    v3[14, 11] := "BsplineEval"(x := v0[11], lut_grid := "NeuroPLC_Weights".w0, lut_table := lut_tmp);
    // φ[12→14]: evaluate LUT (table offset 6060)
    FOR k := 0 TO 14 DO
        lut_tmp[k] := "NeuroPLC_Weights".w1[6060 + k];
    END_FOR;
    v3[14, 12] := "BsplineEval"(x := v0[12], lut_grid := "NeuroPLC_Weights".w0, lut_table := lut_tmp);
    // φ[13→14]: evaluate LUT (table offset 6075)
    FOR k := 0 TO 14 DO
        lut_tmp[k] := "NeuroPLC_Weights".w1[6075 + k];
    END_FOR;
    v3[14, 13] := "BsplineEval"(x := v0[13], lut_grid := "NeuroPLC_Weights".w0, lut_table := lut_tmp);
    // φ[14→14]: evaluate LUT (table offset 6090)
    FOR k := 0 TO 14 DO
        lut_tmp[k] := "NeuroPLC_Weights".w1[6090 + k];
    END_FOR;
    v3[14, 14] := "BsplineEval"(x := v0[14], lut_grid := "NeuroPLC_Weights".w0, lut_table := lut_tmp);
    // φ[15→14]: evaluate LUT (table offset 6105)
    FOR k := 0 TO 14 DO
        lut_tmp[k] := "NeuroPLC_Weights".w1[6105 + k];
    END_FOR;
    v3[14, 15] := "BsplineEval"(x := v0[15], lut_grid := "NeuroPLC_Weights".w0, lut_table := lut_tmp);
    // φ[16→14]: evaluate LUT (table offset 6120)
    FOR k := 0 TO 14 DO
        lut_tmp[k] := "NeuroPLC_Weights".w1[6120 + k];
    END_FOR;
    v3[14, 16] := "BsplineEval"(x := v0[16], lut_grid := "NeuroPLC_Weights".w0, lut_table := lut_tmp);
    // φ[17→14]: evaluate LUT (table offset 6135)
    FOR k := 0 TO 14 DO
        lut_tmp[k] := "NeuroPLC_Weights".w1[6135 + k];
    END_FOR;
    v3[14, 17] := "BsplineEval"(x := v0[17], lut_grid := "NeuroPLC_Weights".w0, lut_table := lut_tmp);
    // φ[18→14]: evaluate LUT (table offset 6150)
    FOR k := 0 TO 14 DO
        lut_tmp[k] := "NeuroPLC_Weights".w1[6150 + k];
    END_FOR;
    v3[14, 18] := "BsplineEval"(x := v0[18], lut_grid := "NeuroPLC_Weights".w0, lut_table := lut_tmp);
    // φ[19→14]: evaluate LUT (table offset 6165)
    FOR k := 0 TO 14 DO
        lut_tmp[k] := "NeuroPLC_Weights".w1[6165 + k];
    END_FOR;
    v3[14, 19] := "BsplineEval"(x := v0[19], lut_grid := "NeuroPLC_Weights".w0, lut_table := lut_tmp);
    // φ[20→14]: evaluate LUT (table offset 6180)
    FOR k := 0 TO 14 DO
        lut_tmp[k] := "NeuroPLC_Weights".w1[6180 + k];
    END_FOR;
    v3[14, 20] := "BsplineEval"(x := v0[20], lut_grid := "NeuroPLC_Weights".w0, lut_table := lut_tmp);
    // φ[21→14]: evaluate LUT (table offset 6195)
    FOR k := 0 TO 14 DO
        lut_tmp[k] := "NeuroPLC_Weights".w1[6195 + k];
    END_FOR;
    v3[14, 21] := "BsplineEval"(x := v0[21], lut_grid := "NeuroPLC_Weights".w0, lut_table := lut_tmp);
    // φ[22→14]: evaluate LUT (table offset 6210)
    FOR k := 0 TO 14 DO
        lut_tmp[k] := "NeuroPLC_Weights".w1[6210 + k];
    END_FOR;
    v3[14, 22] := "BsplineEval"(x := v0[22], lut_grid := "NeuroPLC_Weights".w0, lut_table := lut_tmp);
    // φ[23→14]: evaluate LUT (table offset 6225)
    FOR k := 0 TO 14 DO
        lut_tmp[k] := "NeuroPLC_Weights".w1[6225 + k];
    END_FOR;
    v3[14, 23] := "BsplineEval"(x := v0[23], lut_grid := "NeuroPLC_Weights".w0, lut_table := lut_tmp);
    // φ[24→14]: evaluate LUT (table offset 6240)
    FOR k := 0 TO 14 DO
        lut_tmp[k] := "NeuroPLC_Weights".w1[6240 + k];
    END_FOR;
    v3[14, 24] := "BsplineEval"(x := v0[24], lut_grid := "NeuroPLC_Weights".w0, lut_table := lut_tmp);
    // φ[25→14]: evaluate LUT (table offset 6255)
    FOR k := 0 TO 14 DO
        lut_tmp[k] := "NeuroPLC_Weights".w1[6255 + k];
    END_FOR;
    v3[14, 25] := "BsplineEval"(x := v0[25], lut_grid := "NeuroPLC_Weights".w0, lut_table := lut_tmp);
    // φ[26→14]: evaluate LUT (table offset 6270)
    FOR k := 0 TO 14 DO
        lut_tmp[k] := "NeuroPLC_Weights".w1[6270 + k];
    END_FOR;
    v3[14, 26] := "BsplineEval"(x := v0[26], lut_grid := "NeuroPLC_Weights".w0, lut_table := lut_tmp);
    // φ[27→14]: evaluate LUT (table offset 6285)
    FOR k := 0 TO 14 DO
        lut_tmp[k] := "NeuroPLC_Weights".w1[6285 + k];
    END_FOR;
    v3[14, 27] := "BsplineEval"(x := v0[27], lut_grid := "NeuroPLC_Weights".w0, lut_table := lut_tmp);
    // φ[0→15]: evaluate LUT (table offset 6300)
    FOR k := 0 TO 14 DO
        lut_tmp[k] := "NeuroPLC_Weights".w1[6300 + k];
    END_FOR;
    v3[15, 0] := "BsplineEval"(x := v0[0], lut_grid := "NeuroPLC_Weights".w0, lut_table := lut_tmp);
    // φ[1→15]: evaluate LUT (table offset 6315)
    FOR k := 0 TO 14 DO
        lut_tmp[k] := "NeuroPLC_Weights".w1[6315 + k];
    END_FOR;
    v3[15, 1] := "BsplineEval"(x := v0[1], lut_grid := "NeuroPLC_Weights".w0, lut_table := lut_tmp);
    // φ[2→15]: evaluate LUT (table offset 6330)
    FOR k := 0 TO 14 DO
        lut_tmp[k] := "NeuroPLC_Weights".w1[6330 + k];
    END_FOR;
    v3[15, 2] := "BsplineEval"(x := v0[2], lut_grid := "NeuroPLC_Weights".w0, lut_table := lut_tmp);
    // φ[3→15]: evaluate LUT (table offset 6345)
    FOR k := 0 TO 14 DO
        lut_tmp[k] := "NeuroPLC_Weights".w1[6345 + k];
    END_FOR;
    v3[15, 3] := "BsplineEval"(x := v0[3], lut_grid := "NeuroPLC_Weights".w0, lut_table := lut_tmp);
    // φ[4→15]: evaluate LUT (table offset 6360)
    FOR k := 0 TO 14 DO
        lut_tmp[k] := "NeuroPLC_Weights".w1[6360 + k];
    END_FOR;
    v3[15, 4] := "BsplineEval"(x := v0[4], lut_grid := "NeuroPLC_Weights".w0, lut_table := lut_tmp);
    // φ[5→15]: evaluate LUT (table offset 6375)
    FOR k := 0 TO 14 DO
        lut_tmp[k] := "NeuroPLC_Weights".w1[6375 + k];
    END_FOR;
    v3[15, 5] := "BsplineEval"(x := v0[5], lut_grid := "NeuroPLC_Weights".w0, lut_table := lut_tmp);
    // φ[6→15]: evaluate LUT (table offset 6390)
    FOR k := 0 TO 14 DO
        lut_tmp[k] := "NeuroPLC_Weights".w1[6390 + k];
    END_FOR;
    v3[15, 6] := "BsplineEval"(x := v0[6], lut_grid := "NeuroPLC_Weights".w0, lut_table := lut_tmp);
    // φ[7→15]: evaluate LUT (table offset 6405)
    FOR k := 0 TO 14 DO
        lut_tmp[k] := "NeuroPLC_Weights".w1[6405 + k];
    END_FOR;
    v3[15, 7] := "BsplineEval"(x := v0[7], lut_grid := "NeuroPLC_Weights".w0, lut_table := lut_tmp);
    // φ[8→15]: evaluate LUT (table offset 6420)
    FOR k := 0 TO 14 DO
        lut_tmp[k] := "NeuroPLC_Weights".w1[6420 + k];
    END_FOR;
    v3[15, 8] := "BsplineEval"(x := v0[8], lut_grid := "NeuroPLC_Weights".w0, lut_table := lut_tmp);
    // φ[9→15]: evaluate LUT (table offset 6435)
    FOR k := 0 TO 14 DO
        lut_tmp[k] := "NeuroPLC_Weights".w1[6435 + k];
    END_FOR;
    v3[15, 9] := "BsplineEval"(x := v0[9], lut_grid := "NeuroPLC_Weights".w0, lut_table := lut_tmp);
    // φ[10→15]: evaluate LUT (table offset 6450)
    FOR k := 0 TO 14 DO
        lut_tmp[k] := "NeuroPLC_Weights".w1[6450 + k];
    END_FOR;
    v3[15, 10] := "BsplineEval"(x := v0[10], lut_grid := "NeuroPLC_Weights".w0, lut_table := lut_tmp);
    // φ[11→15]: evaluate LUT (table offset 6465)
    FOR k := 0 TO 14 DO
        lut_tmp[k] := "NeuroPLC_Weights".w1[6465 + k];
    END_FOR;
    v3[15, 11] := "BsplineEval"(x := v0[11], lut_grid := "NeuroPLC_Weights".w0, lut_table := lut_tmp);
    // φ[12→15]: evaluate LUT (table offset 6480)
    FOR k := 0 TO 14 DO
        lut_tmp[k] := "NeuroPLC_Weights".w1[6480 + k];
    END_FOR;
    v3[15, 12] := "BsplineEval"(x := v0[12], lut_grid := "NeuroPLC_Weights".w0, lut_table := lut_tmp);
    // φ[13→15]: evaluate LUT (table offset 6495)
    FOR k := 0 TO 14 DO
        lut_tmp[k] := "NeuroPLC_Weights".w1[6495 + k];
    END_FOR;
    v3[15, 13] := "BsplineEval"(x := v0[13], lut_grid := "NeuroPLC_Weights".w0, lut_table := lut_tmp);
    // φ[14→15]: evaluate LUT (table offset 6510)
    FOR k := 0 TO 14 DO
        lut_tmp[k] := "NeuroPLC_Weights".w1[6510 + k];
    END_FOR;
    v3[15, 14] := "BsplineEval"(x := v0[14], lut_grid := "NeuroPLC_Weights".w0, lut_table := lut_tmp);
    // φ[15→15]: evaluate LUT (table offset 6525)
    FOR k := 0 TO 14 DO
        lut_tmp[k] := "NeuroPLC_Weights".w1[6525 + k];
    END_FOR;
    v3[15, 15] := "BsplineEval"(x := v0[15], lut_grid := "NeuroPLC_Weights".w0, lut_table := lut_tmp);
    // φ[16→15]: evaluate LUT (table offset 6540)
    FOR k := 0 TO 14 DO
        lut_tmp[k] := "NeuroPLC_Weights".w1[6540 + k];
    END_FOR;
    v3[15, 16] := "BsplineEval"(x := v0[16], lut_grid := "NeuroPLC_Weights".w0, lut_table := lut_tmp);
    // φ[17→15]: evaluate LUT (table offset 6555)
    FOR k := 0 TO 14 DO
        lut_tmp[k] := "NeuroPLC_Weights".w1[6555 + k];
    END_FOR;
    v3[15, 17] := "BsplineEval"(x := v0[17], lut_grid := "NeuroPLC_Weights".w0, lut_table := lut_tmp);
    // φ[18→15]: evaluate LUT (table offset 6570)
    FOR k := 0 TO 14 DO
        lut_tmp[k] := "NeuroPLC_Weights".w1[6570 + k];
    END_FOR;
    v3[15, 18] := "BsplineEval"(x := v0[18], lut_grid := "NeuroPLC_Weights".w0, lut_table := lut_tmp);
    // φ[19→15]: evaluate LUT (table offset 6585)
    FOR k := 0 TO 14 DO
        lut_tmp[k] := "NeuroPLC_Weights".w1[6585 + k];
    END_FOR;
    v3[15, 19] := "BsplineEval"(x := v0[19], lut_grid := "NeuroPLC_Weights".w0, lut_table := lut_tmp);
    // φ[20→15]: evaluate LUT (table offset 6600)
    FOR k := 0 TO 14 DO
        lut_tmp[k] := "NeuroPLC_Weights".w1[6600 + k];
    END_FOR;
    v3[15, 20] := "BsplineEval"(x := v0[20], lut_grid := "NeuroPLC_Weights".w0, lut_table := lut_tmp);
    // φ[21→15]: evaluate LUT (table offset 6615)
    FOR k := 0 TO 14 DO
        lut_tmp[k] := "NeuroPLC_Weights".w1[6615 + k];
    END_FOR;
    v3[15, 21] := "BsplineEval"(x := v0[21], lut_grid := "NeuroPLC_Weights".w0, lut_table := lut_tmp);
    // φ[22→15]: evaluate LUT (table offset 6630)
    FOR k := 0 TO 14 DO
        lut_tmp[k] := "NeuroPLC_Weights".w1[6630 + k];
    END_FOR;
    v3[15, 22] := "BsplineEval"(x := v0[22], lut_grid := "NeuroPLC_Weights".w0, lut_table := lut_tmp);
    // φ[23→15]: evaluate LUT (table offset 6645)
    FOR k := 0 TO 14 DO
        lut_tmp[k] := "NeuroPLC_Weights".w1[6645 + k];
    END_FOR;
    v3[15, 23] := "BsplineEval"(x := v0[23], lut_grid := "NeuroPLC_Weights".w0, lut_table := lut_tmp);
    // φ[24→15]: evaluate LUT (table offset 6660)
    FOR k := 0 TO 14 DO
        lut_tmp[k] := "NeuroPLC_Weights".w1[6660 + k];
    END_FOR;
    v3[15, 24] := "BsplineEval"(x := v0[24], lut_grid := "NeuroPLC_Weights".w0, lut_table := lut_tmp);
    // φ[25→15]: evaluate LUT (table offset 6675)
    FOR k := 0 TO 14 DO
        lut_tmp[k] := "NeuroPLC_Weights".w1[6675 + k];
    END_FOR;
    v3[15, 25] := "BsplineEval"(x := v0[25], lut_grid := "NeuroPLC_Weights".w0, lut_table := lut_tmp);
    // φ[26→15]: evaluate LUT (table offset 6690)
    FOR k := 0 TO 14 DO
        lut_tmp[k] := "NeuroPLC_Weights".w1[6690 + k];
    END_FOR;
    v3[15, 26] := "BsplineEval"(x := v0[26], lut_grid := "NeuroPLC_Weights".w0, lut_table := lut_tmp);
    // φ[27→15]: evaluate LUT (table offset 6705)
    FOR k := 0 TO 14 DO
        lut_tmp[k] := "NeuroPLC_Weights".w1[6705 + k];
    END_FOR;
    v3[15, 27] := "BsplineEval"(x := v0[27], lut_grid := "NeuroPLC_Weights".w0, lut_table := lut_tmp);

    // ---- l0_base: MatMul(28→16) ----
    // W = "NeuroPLC_Weights".w2[:448],   b = w2[448:]
    v2[0] := "NeuroPLC_Weights".w2[448 + 0] + "NeuroPLC_Weights".w2[0] * v1[0] + "NeuroPLC_Weights".w2[1] * v1[1] + "NeuroPLC_Weights".w2[2] * v1[2] + "NeuroPLC_Weights".w2[3] * v1[3] + "NeuroPLC_Weights".w2[4] * v1[4] + "NeuroPLC_Weights".w2[5] * v1[5] + "NeuroPLC_Weights".w2[6] * v1[6] + "NeuroPLC_Weights".w2[7] * v1[7] + "NeuroPLC_Weights".w2[8] * v1[8] + "NeuroPLC_Weights".w2[9] * v1[9] + "NeuroPLC_Weights".w2[10] * v1[10] + "NeuroPLC_Weights".w2[11] * v1[11] + "NeuroPLC_Weights".w2[12] * v1[12] + "NeuroPLC_Weights".w2[13] * v1[13] + "NeuroPLC_Weights".w2[14] * v1[14] + "NeuroPLC_Weights".w2[15] * v1[15] + "NeuroPLC_Weights".w2[16] * v1[16] + "NeuroPLC_Weights".w2[17] * v1[17] + "NeuroPLC_Weights".w2[18] * v1[18] + "NeuroPLC_Weights".w2[19] * v1[19] + "NeuroPLC_Weights".w2[20] * v1[20] + "NeuroPLC_Weights".w2[21] * v1[21] + "NeuroPLC_Weights".w2[22] * v1[22] + "NeuroPLC_Weights".w2[23] * v1[23] + "NeuroPLC_Weights".w2[24] * v1[24] + "NeuroPLC_Weights".w2[25] * v1[25] + "NeuroPLC_Weights".w2[26] * v1[26] + "NeuroPLC_Weights".w2[27] * v1[27];
    v2[1] := "NeuroPLC_Weights".w2[448 + 1] + "NeuroPLC_Weights".w2[28] * v1[0] + "NeuroPLC_Weights".w2[29] * v1[1] + "NeuroPLC_Weights".w2[30] * v1[2] + "NeuroPLC_Weights".w2[31] * v1[3] + "NeuroPLC_Weights".w2[32] * v1[4] + "NeuroPLC_Weights".w2[33] * v1[5] + "NeuroPLC_Weights".w2[34] * v1[6] + "NeuroPLC_Weights".w2[35] * v1[7] + "NeuroPLC_Weights".w2[36] * v1[8] + "NeuroPLC_Weights".w2[37] * v1[9] + "NeuroPLC_Weights".w2[38] * v1[10] + "NeuroPLC_Weights".w2[39] * v1[11] + "NeuroPLC_Weights".w2[40] * v1[12] + "NeuroPLC_Weights".w2[41] * v1[13] + "NeuroPLC_Weights".w2[42] * v1[14] + "NeuroPLC_Weights".w2[43] * v1[15] + "NeuroPLC_Weights".w2[44] * v1[16] + "NeuroPLC_Weights".w2[45] * v1[17] + "NeuroPLC_Weights".w2[46] * v1[18] + "NeuroPLC_Weights".w2[47] * v1[19] + "NeuroPLC_Weights".w2[48] * v1[20] + "NeuroPLC_Weights".w2[49] * v1[21] + "NeuroPLC_Weights".w2[50] * v1[22] + "NeuroPLC_Weights".w2[51] * v1[23] + "NeuroPLC_Weights".w2[52] * v1[24] + "NeuroPLC_Weights".w2[53] * v1[25] + "NeuroPLC_Weights".w2[54] * v1[26] + "NeuroPLC_Weights".w2[55] * v1[27];
    v2[2] := "NeuroPLC_Weights".w2[448 + 2] + "NeuroPLC_Weights".w2[56] * v1[0] + "NeuroPLC_Weights".w2[57] * v1[1] + "NeuroPLC_Weights".w2[58] * v1[2] + "NeuroPLC_Weights".w2[59] * v1[3] + "NeuroPLC_Weights".w2[60] * v1[4] + "NeuroPLC_Weights".w2[61] * v1[5] + "NeuroPLC_Weights".w2[62] * v1[6] + "NeuroPLC_Weights".w2[63] * v1[7] + "NeuroPLC_Weights".w2[64] * v1[8] + "NeuroPLC_Weights".w2[65] * v1[9] + "NeuroPLC_Weights".w2[66] * v1[10] + "NeuroPLC_Weights".w2[67] * v1[11] + "NeuroPLC_Weights".w2[68] * v1[12] + "NeuroPLC_Weights".w2[69] * v1[13] + "NeuroPLC_Weights".w2[70] * v1[14] + "NeuroPLC_Weights".w2[71] * v1[15] + "NeuroPLC_Weights".w2[72] * v1[16] + "NeuroPLC_Weights".w2[73] * v1[17] + "NeuroPLC_Weights".w2[74] * v1[18] + "NeuroPLC_Weights".w2[75] * v1[19] + "NeuroPLC_Weights".w2[76] * v1[20] + "NeuroPLC_Weights".w2[77] * v1[21] + "NeuroPLC_Weights".w2[78] * v1[22] + "NeuroPLC_Weights".w2[79] * v1[23] + "NeuroPLC_Weights".w2[80] * v1[24] + "NeuroPLC_Weights".w2[81] * v1[25] + "NeuroPLC_Weights".w2[82] * v1[26] + "NeuroPLC_Weights".w2[83] * v1[27];
    v2[3] := "NeuroPLC_Weights".w2[448 + 3] + "NeuroPLC_Weights".w2[84] * v1[0] + "NeuroPLC_Weights".w2[85] * v1[1] + "NeuroPLC_Weights".w2[86] * v1[2] + "NeuroPLC_Weights".w2[87] * v1[3] + "NeuroPLC_Weights".w2[88] * v1[4] + "NeuroPLC_Weights".w2[89] * v1[5] + "NeuroPLC_Weights".w2[90] * v1[6] + "NeuroPLC_Weights".w2[91] * v1[7] + "NeuroPLC_Weights".w2[92] * v1[8] + "NeuroPLC_Weights".w2[93] * v1[9] + "NeuroPLC_Weights".w2[94] * v1[10] + "NeuroPLC_Weights".w2[95] * v1[11] + "NeuroPLC_Weights".w2[96] * v1[12] + "NeuroPLC_Weights".w2[97] * v1[13] + "NeuroPLC_Weights".w2[98] * v1[14] + "NeuroPLC_Weights".w2[99] * v1[15] + "NeuroPLC_Weights".w2[100] * v1[16] + "NeuroPLC_Weights".w2[101] * v1[17] + "NeuroPLC_Weights".w2[102] * v1[18] + "NeuroPLC_Weights".w2[103] * v1[19] + "NeuroPLC_Weights".w2[104] * v1[20] + "NeuroPLC_Weights".w2[105] * v1[21] + "NeuroPLC_Weights".w2[106] * v1[22] + "NeuroPLC_Weights".w2[107] * v1[23] + "NeuroPLC_Weights".w2[108] * v1[24] + "NeuroPLC_Weights".w2[109] * v1[25] + "NeuroPLC_Weights".w2[110] * v1[26] + "NeuroPLC_Weights".w2[111] * v1[27];
    v2[4] := "NeuroPLC_Weights".w2[448 + 4] + "NeuroPLC_Weights".w2[112] * v1[0] + "NeuroPLC_Weights".w2[113] * v1[1] + "NeuroPLC_Weights".w2[114] * v1[2] + "NeuroPLC_Weights".w2[115] * v1[3] + "NeuroPLC_Weights".w2[116] * v1[4] + "NeuroPLC_Weights".w2[117] * v1[5] + "NeuroPLC_Weights".w2[118] * v1[6] + "NeuroPLC_Weights".w2[119] * v1[7] + "NeuroPLC_Weights".w2[120] * v1[8] + "NeuroPLC_Weights".w2[121] * v1[9] + "NeuroPLC_Weights".w2[122] * v1[10] + "NeuroPLC_Weights".w2[123] * v1[11] + "NeuroPLC_Weights".w2[124] * v1[12] + "NeuroPLC_Weights".w2[125] * v1[13] + "NeuroPLC_Weights".w2[126] * v1[14] + "NeuroPLC_Weights".w2[127] * v1[15] + "NeuroPLC_Weights".w2[128] * v1[16] + "NeuroPLC_Weights".w2[129] * v1[17] + "NeuroPLC_Weights".w2[130] * v1[18] + "NeuroPLC_Weights".w2[131] * v1[19] + "NeuroPLC_Weights".w2[132] * v1[20] + "NeuroPLC_Weights".w2[133] * v1[21] + "NeuroPLC_Weights".w2[134] * v1[22] + "NeuroPLC_Weights".w2[135] * v1[23] + "NeuroPLC_Weights".w2[136] * v1[24] + "NeuroPLC_Weights".w2[137] * v1[25] + "NeuroPLC_Weights".w2[138] * v1[26] + "NeuroPLC_Weights".w2[139] * v1[27];
    v2[5] := "NeuroPLC_Weights".w2[448 + 5] + "NeuroPLC_Weights".w2[140] * v1[0] + "NeuroPLC_Weights".w2[141] * v1[1] + "NeuroPLC_Weights".w2[142] * v1[2] + "NeuroPLC_Weights".w2[143] * v1[3] + "NeuroPLC_Weights".w2[144] * v1[4] + "NeuroPLC_Weights".w2[145] * v1[5] + "NeuroPLC_Weights".w2[146] * v1[6] + "NeuroPLC_Weights".w2[147] * v1[7] + "NeuroPLC_Weights".w2[148] * v1[8] + "NeuroPLC_Weights".w2[149] * v1[9] + "NeuroPLC_Weights".w2[150] * v1[10] + "NeuroPLC_Weights".w2[151] * v1[11] + "NeuroPLC_Weights".w2[152] * v1[12] + "NeuroPLC_Weights".w2[153] * v1[13] + "NeuroPLC_Weights".w2[154] * v1[14] + "NeuroPLC_Weights".w2[155] * v1[15] + "NeuroPLC_Weights".w2[156] * v1[16] + "NeuroPLC_Weights".w2[157] * v1[17] + "NeuroPLC_Weights".w2[158] * v1[18] + "NeuroPLC_Weights".w2[159] * v1[19] + "NeuroPLC_Weights".w2[160] * v1[20] + "NeuroPLC_Weights".w2[161] * v1[21] + "NeuroPLC_Weights".w2[162] * v1[22] + "NeuroPLC_Weights".w2[163] * v1[23] + "NeuroPLC_Weights".w2[164] * v1[24] + "NeuroPLC_Weights".w2[165] * v1[25] + "NeuroPLC_Weights".w2[166] * v1[26] + "NeuroPLC_Weights".w2[167] * v1[27];
    v2[6] := "NeuroPLC_Weights".w2[448 + 6] + "NeuroPLC_Weights".w2[168] * v1[0] + "NeuroPLC_Weights".w2[169] * v1[1] + "NeuroPLC_Weights".w2[170] * v1[2] + "NeuroPLC_Weights".w2[171] * v1[3] + "NeuroPLC_Weights".w2[172] * v1[4] + "NeuroPLC_Weights".w2[173] * v1[5] + "NeuroPLC_Weights".w2[174] * v1[6] + "NeuroPLC_Weights".w2[175] * v1[7] + "NeuroPLC_Weights".w2[176] * v1[8] + "NeuroPLC_Weights".w2[177] * v1[9] + "NeuroPLC_Weights".w2[178] * v1[10] + "NeuroPLC_Weights".w2[179] * v1[11] + "NeuroPLC_Weights".w2[180] * v1[12] + "NeuroPLC_Weights".w2[181] * v1[13] + "NeuroPLC_Weights".w2[182] * v1[14] + "NeuroPLC_Weights".w2[183] * v1[15] + "NeuroPLC_Weights".w2[184] * v1[16] + "NeuroPLC_Weights".w2[185] * v1[17] + "NeuroPLC_Weights".w2[186] * v1[18] + "NeuroPLC_Weights".w2[187] * v1[19] + "NeuroPLC_Weights".w2[188] * v1[20] + "NeuroPLC_Weights".w2[189] * v1[21] + "NeuroPLC_Weights".w2[190] * v1[22] + "NeuroPLC_Weights".w2[191] * v1[23] + "NeuroPLC_Weights".w2[192] * v1[24] + "NeuroPLC_Weights".w2[193] * v1[25] + "NeuroPLC_Weights".w2[194] * v1[26] + "NeuroPLC_Weights".w2[195] * v1[27];
    v2[7] := "NeuroPLC_Weights".w2[448 + 7] + "NeuroPLC_Weights".w2[196] * v1[0] + "NeuroPLC_Weights".w2[197] * v1[1] + "NeuroPLC_Weights".w2[198] * v1[2] + "NeuroPLC_Weights".w2[199] * v1[3] + "NeuroPLC_Weights".w2[200] * v1[4] + "NeuroPLC_Weights".w2[201] * v1[5] + "NeuroPLC_Weights".w2[202] * v1[6] + "NeuroPLC_Weights".w2[203] * v1[7] + "NeuroPLC_Weights".w2[204] * v1[8] + "NeuroPLC_Weights".w2[205] * v1[9] + "NeuroPLC_Weights".w2[206] * v1[10] + "NeuroPLC_Weights".w2[207] * v1[11] + "NeuroPLC_Weights".w2[208] * v1[12] + "NeuroPLC_Weights".w2[209] * v1[13] + "NeuroPLC_Weights".w2[210] * v1[14] + "NeuroPLC_Weights".w2[211] * v1[15] + "NeuroPLC_Weights".w2[212] * v1[16] + "NeuroPLC_Weights".w2[213] * v1[17] + "NeuroPLC_Weights".w2[214] * v1[18] + "NeuroPLC_Weights".w2[215] * v1[19] + "NeuroPLC_Weights".w2[216] * v1[20] + "NeuroPLC_Weights".w2[217] * v1[21] + "NeuroPLC_Weights".w2[218] * v1[22] + "NeuroPLC_Weights".w2[219] * v1[23] + "NeuroPLC_Weights".w2[220] * v1[24] + "NeuroPLC_Weights".w2[221] * v1[25] + "NeuroPLC_Weights".w2[222] * v1[26] + "NeuroPLC_Weights".w2[223] * v1[27];
    v2[8] := "NeuroPLC_Weights".w2[448 + 8] + "NeuroPLC_Weights".w2[224] * v1[0] + "NeuroPLC_Weights".w2[225] * v1[1] + "NeuroPLC_Weights".w2[226] * v1[2] + "NeuroPLC_Weights".w2[227] * v1[3] + "NeuroPLC_Weights".w2[228] * v1[4] + "NeuroPLC_Weights".w2[229] * v1[5] + "NeuroPLC_Weights".w2[230] * v1[6] + "NeuroPLC_Weights".w2[231] * v1[7] + "NeuroPLC_Weights".w2[232] * v1[8] + "NeuroPLC_Weights".w2[233] * v1[9] + "NeuroPLC_Weights".w2[234] * v1[10] + "NeuroPLC_Weights".w2[235] * v1[11] + "NeuroPLC_Weights".w2[236] * v1[12] + "NeuroPLC_Weights".w2[237] * v1[13] + "NeuroPLC_Weights".w2[238] * v1[14] + "NeuroPLC_Weights".w2[239] * v1[15] + "NeuroPLC_Weights".w2[240] * v1[16] + "NeuroPLC_Weights".w2[241] * v1[17] + "NeuroPLC_Weights".w2[242] * v1[18] + "NeuroPLC_Weights".w2[243] * v1[19] + "NeuroPLC_Weights".w2[244] * v1[20] + "NeuroPLC_Weights".w2[245] * v1[21] + "NeuroPLC_Weights".w2[246] * v1[22] + "NeuroPLC_Weights".w2[247] * v1[23] + "NeuroPLC_Weights".w2[248] * v1[24] + "NeuroPLC_Weights".w2[249] * v1[25] + "NeuroPLC_Weights".w2[250] * v1[26] + "NeuroPLC_Weights".w2[251] * v1[27];
    v2[9] := "NeuroPLC_Weights".w2[448 + 9] + "NeuroPLC_Weights".w2[252] * v1[0] + "NeuroPLC_Weights".w2[253] * v1[1] + "NeuroPLC_Weights".w2[254] * v1[2] + "NeuroPLC_Weights".w2[255] * v1[3] + "NeuroPLC_Weights".w2[256] * v1[4] + "NeuroPLC_Weights".w2[257] * v1[5] + "NeuroPLC_Weights".w2[258] * v1[6] + "NeuroPLC_Weights".w2[259] * v1[7] + "NeuroPLC_Weights".w2[260] * v1[8] + "NeuroPLC_Weights".w2[261] * v1[9] + "NeuroPLC_Weights".w2[262] * v1[10] + "NeuroPLC_Weights".w2[263] * v1[11] + "NeuroPLC_Weights".w2[264] * v1[12] + "NeuroPLC_Weights".w2[265] * v1[13] + "NeuroPLC_Weights".w2[266] * v1[14] + "NeuroPLC_Weights".w2[267] * v1[15] + "NeuroPLC_Weights".w2[268] * v1[16] + "NeuroPLC_Weights".w2[269] * v1[17] + "NeuroPLC_Weights".w2[270] * v1[18] + "NeuroPLC_Weights".w2[271] * v1[19] + "NeuroPLC_Weights".w2[272] * v1[20] + "NeuroPLC_Weights".w2[273] * v1[21] + "NeuroPLC_Weights".w2[274] * v1[22] + "NeuroPLC_Weights".w2[275] * v1[23] + "NeuroPLC_Weights".w2[276] * v1[24] + "NeuroPLC_Weights".w2[277] * v1[25] + "NeuroPLC_Weights".w2[278] * v1[26] + "NeuroPLC_Weights".w2[279] * v1[27];
    v2[10] := "NeuroPLC_Weights".w2[448 + 10] + "NeuroPLC_Weights".w2[280] * v1[0] + "NeuroPLC_Weights".w2[281] * v1[1] + "NeuroPLC_Weights".w2[282] * v1[2] + "NeuroPLC_Weights".w2[283] * v1[3] + "NeuroPLC_Weights".w2[284] * v1[4] + "NeuroPLC_Weights".w2[285] * v1[5] + "NeuroPLC_Weights".w2[286] * v1[6] + "NeuroPLC_Weights".w2[287] * v1[7] + "NeuroPLC_Weights".w2[288] * v1[8] + "NeuroPLC_Weights".w2[289] * v1[9] + "NeuroPLC_Weights".w2[290] * v1[10] + "NeuroPLC_Weights".w2[291] * v1[11] + "NeuroPLC_Weights".w2[292] * v1[12] + "NeuroPLC_Weights".w2[293] * v1[13] + "NeuroPLC_Weights".w2[294] * v1[14] + "NeuroPLC_Weights".w2[295] * v1[15] + "NeuroPLC_Weights".w2[296] * v1[16] + "NeuroPLC_Weights".w2[297] * v1[17] + "NeuroPLC_Weights".w2[298] * v1[18] + "NeuroPLC_Weights".w2[299] * v1[19] + "NeuroPLC_Weights".w2[300] * v1[20] + "NeuroPLC_Weights".w2[301] * v1[21] + "NeuroPLC_Weights".w2[302] * v1[22] + "NeuroPLC_Weights".w2[303] * v1[23] + "NeuroPLC_Weights".w2[304] * v1[24] + "NeuroPLC_Weights".w2[305] * v1[25] + "NeuroPLC_Weights".w2[306] * v1[26] + "NeuroPLC_Weights".w2[307] * v1[27];
    v2[11] := "NeuroPLC_Weights".w2[448 + 11] + "NeuroPLC_Weights".w2[308] * v1[0] + "NeuroPLC_Weights".w2[309] * v1[1] + "NeuroPLC_Weights".w2[310] * v1[2] + "NeuroPLC_Weights".w2[311] * v1[3] + "NeuroPLC_Weights".w2[312] * v1[4] + "NeuroPLC_Weights".w2[313] * v1[5] + "NeuroPLC_Weights".w2[314] * v1[6] + "NeuroPLC_Weights".w2[315] * v1[7] + "NeuroPLC_Weights".w2[316] * v1[8] + "NeuroPLC_Weights".w2[317] * v1[9] + "NeuroPLC_Weights".w2[318] * v1[10] + "NeuroPLC_Weights".w2[319] * v1[11] + "NeuroPLC_Weights".w2[320] * v1[12] + "NeuroPLC_Weights".w2[321] * v1[13] + "NeuroPLC_Weights".w2[322] * v1[14] + "NeuroPLC_Weights".w2[323] * v1[15] + "NeuroPLC_Weights".w2[324] * v1[16] + "NeuroPLC_Weights".w2[325] * v1[17] + "NeuroPLC_Weights".w2[326] * v1[18] + "NeuroPLC_Weights".w2[327] * v1[19] + "NeuroPLC_Weights".w2[328] * v1[20] + "NeuroPLC_Weights".w2[329] * v1[21] + "NeuroPLC_Weights".w2[330] * v1[22] + "NeuroPLC_Weights".w2[331] * v1[23] + "NeuroPLC_Weights".w2[332] * v1[24] + "NeuroPLC_Weights".w2[333] * v1[25] + "NeuroPLC_Weights".w2[334] * v1[26] + "NeuroPLC_Weights".w2[335] * v1[27];
    v2[12] := "NeuroPLC_Weights".w2[448 + 12] + "NeuroPLC_Weights".w2[336] * v1[0] + "NeuroPLC_Weights".w2[337] * v1[1] + "NeuroPLC_Weights".w2[338] * v1[2] + "NeuroPLC_Weights".w2[339] * v1[3] + "NeuroPLC_Weights".w2[340] * v1[4] + "NeuroPLC_Weights".w2[341] * v1[5] + "NeuroPLC_Weights".w2[342] * v1[6] + "NeuroPLC_Weights".w2[343] * v1[7] + "NeuroPLC_Weights".w2[344] * v1[8] + "NeuroPLC_Weights".w2[345] * v1[9] + "NeuroPLC_Weights".w2[346] * v1[10] + "NeuroPLC_Weights".w2[347] * v1[11] + "NeuroPLC_Weights".w2[348] * v1[12] + "NeuroPLC_Weights".w2[349] * v1[13] + "NeuroPLC_Weights".w2[350] * v1[14] + "NeuroPLC_Weights".w2[351] * v1[15] + "NeuroPLC_Weights".w2[352] * v1[16] + "NeuroPLC_Weights".w2[353] * v1[17] + "NeuroPLC_Weights".w2[354] * v1[18] + "NeuroPLC_Weights".w2[355] * v1[19] + "NeuroPLC_Weights".w2[356] * v1[20] + "NeuroPLC_Weights".w2[357] * v1[21] + "NeuroPLC_Weights".w2[358] * v1[22] + "NeuroPLC_Weights".w2[359] * v1[23] + "NeuroPLC_Weights".w2[360] * v1[24] + "NeuroPLC_Weights".w2[361] * v1[25] + "NeuroPLC_Weights".w2[362] * v1[26] + "NeuroPLC_Weights".w2[363] * v1[27];
    v2[13] := "NeuroPLC_Weights".w2[448 + 13] + "NeuroPLC_Weights".w2[364] * v1[0] + "NeuroPLC_Weights".w2[365] * v1[1] + "NeuroPLC_Weights".w2[366] * v1[2] + "NeuroPLC_Weights".w2[367] * v1[3] + "NeuroPLC_Weights".w2[368] * v1[4] + "NeuroPLC_Weights".w2[369] * v1[5] + "NeuroPLC_Weights".w2[370] * v1[6] + "NeuroPLC_Weights".w2[371] * v1[7] + "NeuroPLC_Weights".w2[372] * v1[8] + "NeuroPLC_Weights".w2[373] * v1[9] + "NeuroPLC_Weights".w2[374] * v1[10] + "NeuroPLC_Weights".w2[375] * v1[11] + "NeuroPLC_Weights".w2[376] * v1[12] + "NeuroPLC_Weights".w2[377] * v1[13] + "NeuroPLC_Weights".w2[378] * v1[14] + "NeuroPLC_Weights".w2[379] * v1[15] + "NeuroPLC_Weights".w2[380] * v1[16] + "NeuroPLC_Weights".w2[381] * v1[17] + "NeuroPLC_Weights".w2[382] * v1[18] + "NeuroPLC_Weights".w2[383] * v1[19] + "NeuroPLC_Weights".w2[384] * v1[20] + "NeuroPLC_Weights".w2[385] * v1[21] + "NeuroPLC_Weights".w2[386] * v1[22] + "NeuroPLC_Weights".w2[387] * v1[23] + "NeuroPLC_Weights".w2[388] * v1[24] + "NeuroPLC_Weights".w2[389] * v1[25] + "NeuroPLC_Weights".w2[390] * v1[26] + "NeuroPLC_Weights".w2[391] * v1[27];
    v2[14] := "NeuroPLC_Weights".w2[448 + 14] + "NeuroPLC_Weights".w2[392] * v1[0] + "NeuroPLC_Weights".w2[393] * v1[1] + "NeuroPLC_Weights".w2[394] * v1[2] + "NeuroPLC_Weights".w2[395] * v1[3] + "NeuroPLC_Weights".w2[396] * v1[4] + "NeuroPLC_Weights".w2[397] * v1[5] + "NeuroPLC_Weights".w2[398] * v1[6] + "NeuroPLC_Weights".w2[399] * v1[7] + "NeuroPLC_Weights".w2[400] * v1[8] + "NeuroPLC_Weights".w2[401] * v1[9] + "NeuroPLC_Weights".w2[402] * v1[10] + "NeuroPLC_Weights".w2[403] * v1[11] + "NeuroPLC_Weights".w2[404] * v1[12] + "NeuroPLC_Weights".w2[405] * v1[13] + "NeuroPLC_Weights".w2[406] * v1[14] + "NeuroPLC_Weights".w2[407] * v1[15] + "NeuroPLC_Weights".w2[408] * v1[16] + "NeuroPLC_Weights".w2[409] * v1[17] + "NeuroPLC_Weights".w2[410] * v1[18] + "NeuroPLC_Weights".w2[411] * v1[19] + "NeuroPLC_Weights".w2[412] * v1[20] + "NeuroPLC_Weights".w2[413] * v1[21] + "NeuroPLC_Weights".w2[414] * v1[22] + "NeuroPLC_Weights".w2[415] * v1[23] + "NeuroPLC_Weights".w2[416] * v1[24] + "NeuroPLC_Weights".w2[417] * v1[25] + "NeuroPLC_Weights".w2[418] * v1[26] + "NeuroPLC_Weights".w2[419] * v1[27];
    v2[15] := "NeuroPLC_Weights".w2[448 + 15] + "NeuroPLC_Weights".w2[420] * v1[0] + "NeuroPLC_Weights".w2[421] * v1[1] + "NeuroPLC_Weights".w2[422] * v1[2] + "NeuroPLC_Weights".w2[423] * v1[3] + "NeuroPLC_Weights".w2[424] * v1[4] + "NeuroPLC_Weights".w2[425] * v1[5] + "NeuroPLC_Weights".w2[426] * v1[6] + "NeuroPLC_Weights".w2[427] * v1[7] + "NeuroPLC_Weights".w2[428] * v1[8] + "NeuroPLC_Weights".w2[429] * v1[9] + "NeuroPLC_Weights".w2[430] * v1[10] + "NeuroPLC_Weights".w2[431] * v1[11] + "NeuroPLC_Weights".w2[432] * v1[12] + "NeuroPLC_Weights".w2[433] * v1[13] + "NeuroPLC_Weights".w2[434] * v1[14] + "NeuroPLC_Weights".w2[435] * v1[15] + "NeuroPLC_Weights".w2[436] * v1[16] + "NeuroPLC_Weights".w2[437] * v1[17] + "NeuroPLC_Weights".w2[438] * v1[18] + "NeuroPLC_Weights".w2[439] * v1[19] + "NeuroPLC_Weights".w2[440] * v1[20] + "NeuroPLC_Weights".w2[441] * v1[21] + "NeuroPLC_Weights".w2[442] * v1[22] + "NeuroPLC_Weights".w2[443] * v1[23] + "NeuroPLC_Weights".w2[444] * v1[24] + "NeuroPLC_Weights".w2[445] * v1[25] + "NeuroPLC_Weights".w2[446] * v1[26] + "NeuroPLC_Weights".w2[447] * v1[27];

    // ---- l0_merge: Add (KAN merge) ----
    v4[0] := v2[0] + v3[0];
    v4[1] := v2[1] + v3[1];
    v4[2] := v2[2] + v3[2];
    v4[3] := v2[3] + v3[3];
    v4[4] := v2[4] + v3[4];
    v4[5] := v2[5] + v3[5];
    v4[6] := v2[6] + v3[6];
    v4[7] := v2[7] + v3[7];
    v4[8] := v2[8] + v3[8];
    v4[9] := v2[9] + v3[9];
    v4[10] := v2[10] + v3[10];
    v4[11] := v2[11] + v3[11];
    v4[12] := v2[12] + v3[12];
    v4[13] := v2[13] + v3[13];
    v4[14] := v2[14] + v3[14];
    v4[15] := v2[15] + v3[15];

    // ---- l1_silu: SILU ----
    v5[0] := v4[0] / (1.0 + EXP(-v4[0]));
    v5[1] := v4[1] / (1.0 + EXP(-v4[1]));
    v5[2] := v4[2] / (1.0 + EXP(-v4[2]));
    v5[3] := v4[3] / (1.0 + EXP(-v4[3]));
    v5[4] := v4[4] / (1.0 + EXP(-v4[4]));
    v5[5] := v4[5] / (1.0 + EXP(-v4[5]));
    v5[6] := v4[6] / (1.0 + EXP(-v4[6]));
    v5[7] := v4[7] / (1.0 + EXP(-v4[7]));
    v5[8] := v4[8] / (1.0 + EXP(-v4[8]));
    v5[9] := v4[9] / (1.0 + EXP(-v4[9]));
    v5[10] := v4[10] / (1.0 + EXP(-v4[10]));
    v5[11] := v4[11] / (1.0 + EXP(-v4[11]));
    v5[12] := v4[12] / (1.0 + EXP(-v4[12]));
    v5[13] := v4[13] / (1.0 + EXP(-v4[13]));
    v5[14] := v4[14] / (1.0 + EXP(-v4[14]));
    v5[15] := v4[15] / (1.0 + EXP(-v4[15]));

    // ---- l1_bspline: BsplineLUT(16×4, 15pts) ----
    // φ[0→0]: evaluate LUT (table offset 0)
    FOR k := 0 TO 14 DO
        lut_tmp[k] := "NeuroPLC_Weights".w4[0 + k];
    END_FOR;
    v7[0, 0] := "BsplineEval"(x := v4[0], lut_grid := "NeuroPLC_Weights".w3, lut_table := lut_tmp);
    // φ[1→0]: evaluate LUT (table offset 15)
    FOR k := 0 TO 14 DO
        lut_tmp[k] := "NeuroPLC_Weights".w4[15 + k];
    END_FOR;
    v7[0, 1] := "BsplineEval"(x := v4[1], lut_grid := "NeuroPLC_Weights".w3, lut_table := lut_tmp);
    // φ[2→0]: evaluate LUT (table offset 30)
    FOR k := 0 TO 14 DO
        lut_tmp[k] := "NeuroPLC_Weights".w4[30 + k];
    END_FOR;
    v7[0, 2] := "BsplineEval"(x := v4[2], lut_grid := "NeuroPLC_Weights".w3, lut_table := lut_tmp);
    // φ[3→0]: evaluate LUT (table offset 45)
    FOR k := 0 TO 14 DO
        lut_tmp[k] := "NeuroPLC_Weights".w4[45 + k];
    END_FOR;
    v7[0, 3] := "BsplineEval"(x := v4[3], lut_grid := "NeuroPLC_Weights".w3, lut_table := lut_tmp);
    // φ[4→0]: evaluate LUT (table offset 60)
    FOR k := 0 TO 14 DO
        lut_tmp[k] := "NeuroPLC_Weights".w4[60 + k];
    END_FOR;
    v7[0, 4] := "BsplineEval"(x := v4[4], lut_grid := "NeuroPLC_Weights".w3, lut_table := lut_tmp);
    // φ[5→0]: evaluate LUT (table offset 75)
    FOR k := 0 TO 14 DO
        lut_tmp[k] := "NeuroPLC_Weights".w4[75 + k];
    END_FOR;
    v7[0, 5] := "BsplineEval"(x := v4[5], lut_grid := "NeuroPLC_Weights".w3, lut_table := lut_tmp);
    // φ[6→0]: evaluate LUT (table offset 90)
    FOR k := 0 TO 14 DO
        lut_tmp[k] := "NeuroPLC_Weights".w4[90 + k];
    END_FOR;
    v7[0, 6] := "BsplineEval"(x := v4[6], lut_grid := "NeuroPLC_Weights".w3, lut_table := lut_tmp);
    // φ[7→0]: evaluate LUT (table offset 105)
    FOR k := 0 TO 14 DO
        lut_tmp[k] := "NeuroPLC_Weights".w4[105 + k];
    END_FOR;
    v7[0, 7] := "BsplineEval"(x := v4[7], lut_grid := "NeuroPLC_Weights".w3, lut_table := lut_tmp);
    // φ[8→0]: evaluate LUT (table offset 120)
    FOR k := 0 TO 14 DO
        lut_tmp[k] := "NeuroPLC_Weights".w4[120 + k];
    END_FOR;
    v7[0, 8] := "BsplineEval"(x := v4[8], lut_grid := "NeuroPLC_Weights".w3, lut_table := lut_tmp);
    // φ[9→0]: evaluate LUT (table offset 135)
    FOR k := 0 TO 14 DO
        lut_tmp[k] := "NeuroPLC_Weights".w4[135 + k];
    END_FOR;
    v7[0, 9] := "BsplineEval"(x := v4[9], lut_grid := "NeuroPLC_Weights".w3, lut_table := lut_tmp);
    // φ[10→0]: evaluate LUT (table offset 150)
    FOR k := 0 TO 14 DO
        lut_tmp[k] := "NeuroPLC_Weights".w4[150 + k];
    END_FOR;
    v7[0, 10] := "BsplineEval"(x := v4[10], lut_grid := "NeuroPLC_Weights".w3, lut_table := lut_tmp);
    // φ[11→0]: evaluate LUT (table offset 165)
    FOR k := 0 TO 14 DO
        lut_tmp[k] := "NeuroPLC_Weights".w4[165 + k];
    END_FOR;
    v7[0, 11] := "BsplineEval"(x := v4[11], lut_grid := "NeuroPLC_Weights".w3, lut_table := lut_tmp);
    // φ[12→0]: evaluate LUT (table offset 180)
    FOR k := 0 TO 14 DO
        lut_tmp[k] := "NeuroPLC_Weights".w4[180 + k];
    END_FOR;
    v7[0, 12] := "BsplineEval"(x := v4[12], lut_grid := "NeuroPLC_Weights".w3, lut_table := lut_tmp);
    // φ[13→0]: evaluate LUT (table offset 195)
    FOR k := 0 TO 14 DO
        lut_tmp[k] := "NeuroPLC_Weights".w4[195 + k];
    END_FOR;
    v7[0, 13] := "BsplineEval"(x := v4[13], lut_grid := "NeuroPLC_Weights".w3, lut_table := lut_tmp);
    // φ[14→0]: evaluate LUT (table offset 210)
    FOR k := 0 TO 14 DO
        lut_tmp[k] := "NeuroPLC_Weights".w4[210 + k];
    END_FOR;
    v7[0, 14] := "BsplineEval"(x := v4[14], lut_grid := "NeuroPLC_Weights".w3, lut_table := lut_tmp);
    // φ[15→0]: evaluate LUT (table offset 225)
    FOR k := 0 TO 14 DO
        lut_tmp[k] := "NeuroPLC_Weights".w4[225 + k];
    END_FOR;
    v7[0, 15] := "BsplineEval"(x := v4[15], lut_grid := "NeuroPLC_Weights".w3, lut_table := lut_tmp);
    // φ[0→1]: evaluate LUT (table offset 240)
    FOR k := 0 TO 14 DO
        lut_tmp[k] := "NeuroPLC_Weights".w4[240 + k];
    END_FOR;
    v7[1, 0] := "BsplineEval"(x := v4[0], lut_grid := "NeuroPLC_Weights".w3, lut_table := lut_tmp);
    // φ[1→1]: evaluate LUT (table offset 255)
    FOR k := 0 TO 14 DO
        lut_tmp[k] := "NeuroPLC_Weights".w4[255 + k];
    END_FOR;
    v7[1, 1] := "BsplineEval"(x := v4[1], lut_grid := "NeuroPLC_Weights".w3, lut_table := lut_tmp);
    // φ[2→1]: evaluate LUT (table offset 270)
    FOR k := 0 TO 14 DO
        lut_tmp[k] := "NeuroPLC_Weights".w4[270 + k];
    END_FOR;
    v7[1, 2] := "BsplineEval"(x := v4[2], lut_grid := "NeuroPLC_Weights".w3, lut_table := lut_tmp);
    // φ[3→1]: evaluate LUT (table offset 285)
    FOR k := 0 TO 14 DO
        lut_tmp[k] := "NeuroPLC_Weights".w4[285 + k];
    END_FOR;
    v7[1, 3] := "BsplineEval"(x := v4[3], lut_grid := "NeuroPLC_Weights".w3, lut_table := lut_tmp);
    // φ[4→1]: evaluate LUT (table offset 300)
    FOR k := 0 TO 14 DO
        lut_tmp[k] := "NeuroPLC_Weights".w4[300 + k];
    END_FOR;
    v7[1, 4] := "BsplineEval"(x := v4[4], lut_grid := "NeuroPLC_Weights".w3, lut_table := lut_tmp);
    // φ[5→1]: evaluate LUT (table offset 315)
    FOR k := 0 TO 14 DO
        lut_tmp[k] := "NeuroPLC_Weights".w4[315 + k];
    END_FOR;
    v7[1, 5] := "BsplineEval"(x := v4[5], lut_grid := "NeuroPLC_Weights".w3, lut_table := lut_tmp);
    // φ[6→1]: evaluate LUT (table offset 330)
    FOR k := 0 TO 14 DO
        lut_tmp[k] := "NeuroPLC_Weights".w4[330 + k];
    END_FOR;
    v7[1, 6] := "BsplineEval"(x := v4[6], lut_grid := "NeuroPLC_Weights".w3, lut_table := lut_tmp);
    // φ[7→1]: evaluate LUT (table offset 345)
    FOR k := 0 TO 14 DO
        lut_tmp[k] := "NeuroPLC_Weights".w4[345 + k];
    END_FOR;
    v7[1, 7] := "BsplineEval"(x := v4[7], lut_grid := "NeuroPLC_Weights".w3, lut_table := lut_tmp);
    // φ[8→1]: evaluate LUT (table offset 360)
    FOR k := 0 TO 14 DO
        lut_tmp[k] := "NeuroPLC_Weights".w4[360 + k];
    END_FOR;
    v7[1, 8] := "BsplineEval"(x := v4[8], lut_grid := "NeuroPLC_Weights".w3, lut_table := lut_tmp);
    // φ[9→1]: evaluate LUT (table offset 375)
    FOR k := 0 TO 14 DO
        lut_tmp[k] := "NeuroPLC_Weights".w4[375 + k];
    END_FOR;
    v7[1, 9] := "BsplineEval"(x := v4[9], lut_grid := "NeuroPLC_Weights".w3, lut_table := lut_tmp);
    // φ[10→1]: evaluate LUT (table offset 390)
    FOR k := 0 TO 14 DO
        lut_tmp[k] := "NeuroPLC_Weights".w4[390 + k];
    END_FOR;
    v7[1, 10] := "BsplineEval"(x := v4[10], lut_grid := "NeuroPLC_Weights".w3, lut_table := lut_tmp);
    // φ[11→1]: evaluate LUT (table offset 405)
    FOR k := 0 TO 14 DO
        lut_tmp[k] := "NeuroPLC_Weights".w4[405 + k];
    END_FOR;
    v7[1, 11] := "BsplineEval"(x := v4[11], lut_grid := "NeuroPLC_Weights".w3, lut_table := lut_tmp);
    // φ[12→1]: evaluate LUT (table offset 420)
    FOR k := 0 TO 14 DO
        lut_tmp[k] := "NeuroPLC_Weights".w4[420 + k];
    END_FOR;
    v7[1, 12] := "BsplineEval"(x := v4[12], lut_grid := "NeuroPLC_Weights".w3, lut_table := lut_tmp);
    // φ[13→1]: evaluate LUT (table offset 435)
    FOR k := 0 TO 14 DO
        lut_tmp[k] := "NeuroPLC_Weights".w4[435 + k];
    END_FOR;
    v7[1, 13] := "BsplineEval"(x := v4[13], lut_grid := "NeuroPLC_Weights".w3, lut_table := lut_tmp);
    // φ[14→1]: evaluate LUT (table offset 450)
    FOR k := 0 TO 14 DO
        lut_tmp[k] := "NeuroPLC_Weights".w4[450 + k];
    END_FOR;
    v7[1, 14] := "BsplineEval"(x := v4[14], lut_grid := "NeuroPLC_Weights".w3, lut_table := lut_tmp);
    // φ[15→1]: evaluate LUT (table offset 465)
    FOR k := 0 TO 14 DO
        lut_tmp[k] := "NeuroPLC_Weights".w4[465 + k];
    END_FOR;
    v7[1, 15] := "BsplineEval"(x := v4[15], lut_grid := "NeuroPLC_Weights".w3, lut_table := lut_tmp);
    // φ[0→2]: evaluate LUT (table offset 480)
    FOR k := 0 TO 14 DO
        lut_tmp[k] := "NeuroPLC_Weights".w4[480 + k];
    END_FOR;
    v7[2, 0] := "BsplineEval"(x := v4[0], lut_grid := "NeuroPLC_Weights".w3, lut_table := lut_tmp);
    // φ[1→2]: evaluate LUT (table offset 495)
    FOR k := 0 TO 14 DO
        lut_tmp[k] := "NeuroPLC_Weights".w4[495 + k];
    END_FOR;
    v7[2, 1] := "BsplineEval"(x := v4[1], lut_grid := "NeuroPLC_Weights".w3, lut_table := lut_tmp);
    // φ[2→2]: evaluate LUT (table offset 510)
    FOR k := 0 TO 14 DO
        lut_tmp[k] := "NeuroPLC_Weights".w4[510 + k];
    END_FOR;
    v7[2, 2] := "BsplineEval"(x := v4[2], lut_grid := "NeuroPLC_Weights".w3, lut_table := lut_tmp);
    // φ[3→2]: evaluate LUT (table offset 525)
    FOR k := 0 TO 14 DO
        lut_tmp[k] := "NeuroPLC_Weights".w4[525 + k];
    END_FOR;
    v7[2, 3] := "BsplineEval"(x := v4[3], lut_grid := "NeuroPLC_Weights".w3, lut_table := lut_tmp);
    // φ[4→2]: evaluate LUT (table offset 540)
    FOR k := 0 TO 14 DO
        lut_tmp[k] := "NeuroPLC_Weights".w4[540 + k];
    END_FOR;
    v7[2, 4] := "BsplineEval"(x := v4[4], lut_grid := "NeuroPLC_Weights".w3, lut_table := lut_tmp);
    // φ[5→2]: evaluate LUT (table offset 555)
    FOR k := 0 TO 14 DO
        lut_tmp[k] := "NeuroPLC_Weights".w4[555 + k];
    END_FOR;
    v7[2, 5] := "BsplineEval"(x := v4[5], lut_grid := "NeuroPLC_Weights".w3, lut_table := lut_tmp);
    // φ[6→2]: evaluate LUT (table offset 570)
    FOR k := 0 TO 14 DO
        lut_tmp[k] := "NeuroPLC_Weights".w4[570 + k];
    END_FOR;
    v7[2, 6] := "BsplineEval"(x := v4[6], lut_grid := "NeuroPLC_Weights".w3, lut_table := lut_tmp);
    // φ[7→2]: evaluate LUT (table offset 585)
    FOR k := 0 TO 14 DO
        lut_tmp[k] := "NeuroPLC_Weights".w4[585 + k];
    END_FOR;
    v7[2, 7] := "BsplineEval"(x := v4[7], lut_grid := "NeuroPLC_Weights".w3, lut_table := lut_tmp);
    // φ[8→2]: evaluate LUT (table offset 600)
    FOR k := 0 TO 14 DO
        lut_tmp[k] := "NeuroPLC_Weights".w4[600 + k];
    END_FOR;
    v7[2, 8] := "BsplineEval"(x := v4[8], lut_grid := "NeuroPLC_Weights".w3, lut_table := lut_tmp);
    // φ[9→2]: evaluate LUT (table offset 615)
    FOR k := 0 TO 14 DO
        lut_tmp[k] := "NeuroPLC_Weights".w4[615 + k];
    END_FOR;
    v7[2, 9] := "BsplineEval"(x := v4[9], lut_grid := "NeuroPLC_Weights".w3, lut_table := lut_tmp);
    // φ[10→2]: evaluate LUT (table offset 630)
    FOR k := 0 TO 14 DO
        lut_tmp[k] := "NeuroPLC_Weights".w4[630 + k];
    END_FOR;
    v7[2, 10] := "BsplineEval"(x := v4[10], lut_grid := "NeuroPLC_Weights".w3, lut_table := lut_tmp);
    // φ[11→2]: evaluate LUT (table offset 645)
    FOR k := 0 TO 14 DO
        lut_tmp[k] := "NeuroPLC_Weights".w4[645 + k];
    END_FOR;
    v7[2, 11] := "BsplineEval"(x := v4[11], lut_grid := "NeuroPLC_Weights".w3, lut_table := lut_tmp);
    // φ[12→2]: evaluate LUT (table offset 660)
    FOR k := 0 TO 14 DO
        lut_tmp[k] := "NeuroPLC_Weights".w4[660 + k];
    END_FOR;
    v7[2, 12] := "BsplineEval"(x := v4[12], lut_grid := "NeuroPLC_Weights".w3, lut_table := lut_tmp);
    // φ[13→2]: evaluate LUT (table offset 675)
    FOR k := 0 TO 14 DO
        lut_tmp[k] := "NeuroPLC_Weights".w4[675 + k];
    END_FOR;
    v7[2, 13] := "BsplineEval"(x := v4[13], lut_grid := "NeuroPLC_Weights".w3, lut_table := lut_tmp);
    // φ[14→2]: evaluate LUT (table offset 690)
    FOR k := 0 TO 14 DO
        lut_tmp[k] := "NeuroPLC_Weights".w4[690 + k];
    END_FOR;
    v7[2, 14] := "BsplineEval"(x := v4[14], lut_grid := "NeuroPLC_Weights".w3, lut_table := lut_tmp);
    // φ[15→2]: evaluate LUT (table offset 705)
    FOR k := 0 TO 14 DO
        lut_tmp[k] := "NeuroPLC_Weights".w4[705 + k];
    END_FOR;
    v7[2, 15] := "BsplineEval"(x := v4[15], lut_grid := "NeuroPLC_Weights".w3, lut_table := lut_tmp);
    // φ[0→3]: evaluate LUT (table offset 720)
    FOR k := 0 TO 14 DO
        lut_tmp[k] := "NeuroPLC_Weights".w4[720 + k];
    END_FOR;
    v7[3, 0] := "BsplineEval"(x := v4[0], lut_grid := "NeuroPLC_Weights".w3, lut_table := lut_tmp);
    // φ[1→3]: evaluate LUT (table offset 735)
    FOR k := 0 TO 14 DO
        lut_tmp[k] := "NeuroPLC_Weights".w4[735 + k];
    END_FOR;
    v7[3, 1] := "BsplineEval"(x := v4[1], lut_grid := "NeuroPLC_Weights".w3, lut_table := lut_tmp);
    // φ[2→3]: evaluate LUT (table offset 750)
    FOR k := 0 TO 14 DO
        lut_tmp[k] := "NeuroPLC_Weights".w4[750 + k];
    END_FOR;
    v7[3, 2] := "BsplineEval"(x := v4[2], lut_grid := "NeuroPLC_Weights".w3, lut_table := lut_tmp);
    // φ[3→3]: evaluate LUT (table offset 765)
    FOR k := 0 TO 14 DO
        lut_tmp[k] := "NeuroPLC_Weights".w4[765 + k];
    END_FOR;
    v7[3, 3] := "BsplineEval"(x := v4[3], lut_grid := "NeuroPLC_Weights".w3, lut_table := lut_tmp);
    // φ[4→3]: evaluate LUT (table offset 780)
    FOR k := 0 TO 14 DO
        lut_tmp[k] := "NeuroPLC_Weights".w4[780 + k];
    END_FOR;
    v7[3, 4] := "BsplineEval"(x := v4[4], lut_grid := "NeuroPLC_Weights".w3, lut_table := lut_tmp);
    // φ[5→3]: evaluate LUT (table offset 795)
    FOR k := 0 TO 14 DO
        lut_tmp[k] := "NeuroPLC_Weights".w4[795 + k];
    END_FOR;
    v7[3, 5] := "BsplineEval"(x := v4[5], lut_grid := "NeuroPLC_Weights".w3, lut_table := lut_tmp);
    // φ[6→3]: evaluate LUT (table offset 810)
    FOR k := 0 TO 14 DO
        lut_tmp[k] := "NeuroPLC_Weights".w4[810 + k];
    END_FOR;
    v7[3, 6] := "BsplineEval"(x := v4[6], lut_grid := "NeuroPLC_Weights".w3, lut_table := lut_tmp);
    // φ[7→3]: evaluate LUT (table offset 825)
    FOR k := 0 TO 14 DO
        lut_tmp[k] := "NeuroPLC_Weights".w4[825 + k];
    END_FOR;
    v7[3, 7] := "BsplineEval"(x := v4[7], lut_grid := "NeuroPLC_Weights".w3, lut_table := lut_tmp);
    // φ[8→3]: evaluate LUT (table offset 840)
    FOR k := 0 TO 14 DO
        lut_tmp[k] := "NeuroPLC_Weights".w4[840 + k];
    END_FOR;
    v7[3, 8] := "BsplineEval"(x := v4[8], lut_grid := "NeuroPLC_Weights".w3, lut_table := lut_tmp);
    // φ[9→3]: evaluate LUT (table offset 855)
    FOR k := 0 TO 14 DO
        lut_tmp[k] := "NeuroPLC_Weights".w4[855 + k];
    END_FOR;
    v7[3, 9] := "BsplineEval"(x := v4[9], lut_grid := "NeuroPLC_Weights".w3, lut_table := lut_tmp);
    // φ[10→3]: evaluate LUT (table offset 870)
    FOR k := 0 TO 14 DO
        lut_tmp[k] := "NeuroPLC_Weights".w4[870 + k];
    END_FOR;
    v7[3, 10] := "BsplineEval"(x := v4[10], lut_grid := "NeuroPLC_Weights".w3, lut_table := lut_tmp);
    // φ[11→3]: evaluate LUT (table offset 885)
    FOR k := 0 TO 14 DO
        lut_tmp[k] := "NeuroPLC_Weights".w4[885 + k];
    END_FOR;
    v7[3, 11] := "BsplineEval"(x := v4[11], lut_grid := "NeuroPLC_Weights".w3, lut_table := lut_tmp);
    // φ[12→3]: evaluate LUT (table offset 900)
    FOR k := 0 TO 14 DO
        lut_tmp[k] := "NeuroPLC_Weights".w4[900 + k];
    END_FOR;
    v7[3, 12] := "BsplineEval"(x := v4[12], lut_grid := "NeuroPLC_Weights".w3, lut_table := lut_tmp);
    // φ[13→3]: evaluate LUT (table offset 915)
    FOR k := 0 TO 14 DO
        lut_tmp[k] := "NeuroPLC_Weights".w4[915 + k];
    END_FOR;
    v7[3, 13] := "BsplineEval"(x := v4[13], lut_grid := "NeuroPLC_Weights".w3, lut_table := lut_tmp);
    // φ[14→3]: evaluate LUT (table offset 930)
    FOR k := 0 TO 14 DO
        lut_tmp[k] := "NeuroPLC_Weights".w4[930 + k];
    END_FOR;
    v7[3, 14] := "BsplineEval"(x := v4[14], lut_grid := "NeuroPLC_Weights".w3, lut_table := lut_tmp);
    // φ[15→3]: evaluate LUT (table offset 945)
    FOR k := 0 TO 14 DO
        lut_tmp[k] := "NeuroPLC_Weights".w4[945 + k];
    END_FOR;
    v7[3, 15] := "BsplineEval"(x := v4[15], lut_grid := "NeuroPLC_Weights".w3, lut_table := lut_tmp);

    // ---- l1_base: MatMul(16→4) ----
    // W = "NeuroPLC_Weights".w5[:64],   b = w5[64:]
    v6[0] := "NeuroPLC_Weights".w5[64 + 0] + "NeuroPLC_Weights".w5[0] * v5[0] + "NeuroPLC_Weights".w5[1] * v5[1] + "NeuroPLC_Weights".w5[2] * v5[2] + "NeuroPLC_Weights".w5[3] * v5[3] + "NeuroPLC_Weights".w5[4] * v5[4] + "NeuroPLC_Weights".w5[5] * v5[5] + "NeuroPLC_Weights".w5[6] * v5[6] + "NeuroPLC_Weights".w5[7] * v5[7] + "NeuroPLC_Weights".w5[8] * v5[8] + "NeuroPLC_Weights".w5[9] * v5[9] + "NeuroPLC_Weights".w5[10] * v5[10] + "NeuroPLC_Weights".w5[11] * v5[11] + "NeuroPLC_Weights".w5[12] * v5[12] + "NeuroPLC_Weights".w5[13] * v5[13] + "NeuroPLC_Weights".w5[14] * v5[14] + "NeuroPLC_Weights".w5[15] * v5[15];
    v6[1] := "NeuroPLC_Weights".w5[64 + 1] + "NeuroPLC_Weights".w5[16] * v5[0] + "NeuroPLC_Weights".w5[17] * v5[1] + "NeuroPLC_Weights".w5[18] * v5[2] + "NeuroPLC_Weights".w5[19] * v5[3] + "NeuroPLC_Weights".w5[20] * v5[4] + "NeuroPLC_Weights".w5[21] * v5[5] + "NeuroPLC_Weights".w5[22] * v5[6] + "NeuroPLC_Weights".w5[23] * v5[7] + "NeuroPLC_Weights".w5[24] * v5[8] + "NeuroPLC_Weights".w5[25] * v5[9] + "NeuroPLC_Weights".w5[26] * v5[10] + "NeuroPLC_Weights".w5[27] * v5[11] + "NeuroPLC_Weights".w5[28] * v5[12] + "NeuroPLC_Weights".w5[29] * v5[13] + "NeuroPLC_Weights".w5[30] * v5[14] + "NeuroPLC_Weights".w5[31] * v5[15];
    v6[2] := "NeuroPLC_Weights".w5[64 + 2] + "NeuroPLC_Weights".w5[32] * v5[0] + "NeuroPLC_Weights".w5[33] * v5[1] + "NeuroPLC_Weights".w5[34] * v5[2] + "NeuroPLC_Weights".w5[35] * v5[3] + "NeuroPLC_Weights".w5[36] * v5[4] + "NeuroPLC_Weights".w5[37] * v5[5] + "NeuroPLC_Weights".w5[38] * v5[6] + "NeuroPLC_Weights".w5[39] * v5[7] + "NeuroPLC_Weights".w5[40] * v5[8] + "NeuroPLC_Weights".w5[41] * v5[9] + "NeuroPLC_Weights".w5[42] * v5[10] + "NeuroPLC_Weights".w5[43] * v5[11] + "NeuroPLC_Weights".w5[44] * v5[12] + "NeuroPLC_Weights".w5[45] * v5[13] + "NeuroPLC_Weights".w5[46] * v5[14] + "NeuroPLC_Weights".w5[47] * v5[15];
    v6[3] := "NeuroPLC_Weights".w5[64 + 3] + "NeuroPLC_Weights".w5[48] * v5[0] + "NeuroPLC_Weights".w5[49] * v5[1] + "NeuroPLC_Weights".w5[50] * v5[2] + "NeuroPLC_Weights".w5[51] * v5[3] + "NeuroPLC_Weights".w5[52] * v5[4] + "NeuroPLC_Weights".w5[53] * v5[5] + "NeuroPLC_Weights".w5[54] * v5[6] + "NeuroPLC_Weights".w5[55] * v5[7] + "NeuroPLC_Weights".w5[56] * v5[8] + "NeuroPLC_Weights".w5[57] * v5[9] + "NeuroPLC_Weights".w5[58] * v5[10] + "NeuroPLC_Weights".w5[59] * v5[11] + "NeuroPLC_Weights".w5[60] * v5[12] + "NeuroPLC_Weights".w5[61] * v5[13] + "NeuroPLC_Weights".w5[62] * v5[14] + "NeuroPLC_Weights".w5[63] * v5[15];

    // ---- l1_merge: Add (KAN merge) ----
    v8[0] := v6[0] + v7[0];
    v8[1] := v6[1] + v7[1];
    v8[2] := v6[2] + v7[2];
    v8[3] := v6[3] + v7[3];

    // ---- softmax: Softmax ----
    softmax_out[0] := EXP(v8[0]);
    softmax_out[1] := EXP(v8[1]);
    softmax_out[2] := EXP(v8[2]);
    softmax_out[3] := EXP(v8[3]);
    sum_val := softmax_out[0]
             + softmax_out[1]
             + softmax_out[2]
             + softmax_out[3]
             ;
    IF sum_val > 0.0 THEN
        softmax_out[0] := softmax_out[0] / sum_val;
        softmax_out[1] := softmax_out[1] / sum_val;
        softmax_out[2] := softmax_out[2] / sum_val;
        softmax_out[3] := softmax_out[3] / sum_val;
    END_IF;

    // ---- Argmax ----
    max_val := softmax_out[0];
    fault_class := 0;
    IF softmax_out[1] > max_val THEN
        max_val := softmax_out[1];
        fault_class := 1;
    END_IF;
    IF softmax_out[2] > max_val THEN
        max_val := softmax_out[2];
        fault_class := 2;
    END_IF;
    IF softmax_out[3] > max_val THEN
        max_val := softmax_out[3];
        fault_class := 3;
    END_IF;
    confidence := max_val;

END_FUNCTION_BLOCK